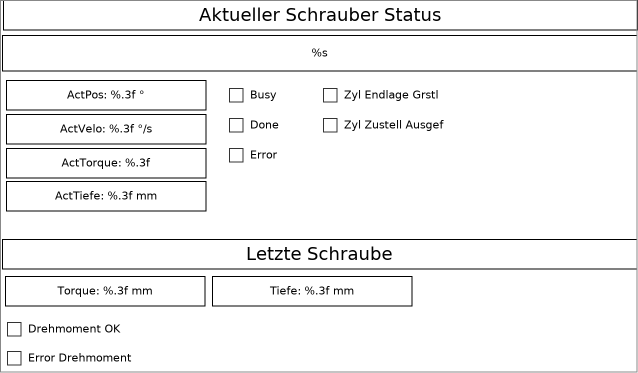
VISUALIZATION Frame_Schrauber_Status  // 638x373
VAR_IN_OUT
	sState	:STRING;
	
	bGrdstlgSchrEinh			: BOOL;
	bZustellZylAusgef			: BOOL;
	
	bBusy	:BOOL;
	bDone	:BOOL;
	bError	:BOOL;
	bErrorDrehmoment		:BOOL;
	bDrehmomentOk			:BOOL;
	nDrehmomentMw			:LREAL;	(* Drehmoment Mittelwert *)
	
	nActPos					:LREAL;
	nActVelo				:LREAL;
	nActTiefe				:LREAL;
	
	nDrehmomentLetzteSchr	:LREAL;	(* Drehmoment Letzte Schraubvorgang *)	
	nTiefeLetzteSchr		:LREAL;	(* Tiefe Letzte Schraubvorgang *)	
END_VAR
    Checkbox (227,80 150x30), "Busy", variable: bBusy, input disabled if: TRUE
    Checkbox (227,110 150x30), "Done", variable: bDone, input disabled if: TRUE
    Checkbox (227,140 150x30), "Error", variable: bError, input disabled if: TRUE
    RoundedRectangle (2,35 635x36), "%s", text variable: sState
    Checkbox (5,314 150x30), "Drehmoment OK", variable: bDrehmomentOk, input disabled if: TRUE
    Rectangle (6,80 200x30), "ActPos: %.3f °", text variable: nActPos
    Rectangle (6,114 200x30), "ActVelo: %.3f °/s", text variable: nActVelo
    Rectangle (6,148 200x30), "ActTorque: %.3f", text variable: nDrehmomentMw
    Rectangle (6,181 200x30), "ActTiefe: %.3f mm", text variable: nActTiefe
    Rectangle (212,276 200x30), "Tiefe: %.3f mm", text variable: nTiefeLetzteSchr
    Rectangle (5,276 200x30), "Torque: %.3f mm", text variable: nDrehmomentLetzteSchr
    Checkbox (5,343 150x30), "Error Drehmoment", variable: bErrorDrehmoment, input disabled if: TRUE
    Rectangle (3,0 635x30), "Aktueller Schrauber Status"
    Rectangle (2,239 635x30), "Letzte Schraube"
    Checkbox (321,80 150x30), "Zyl Endlage Grstl", variable: bGrdstlgSchrEinh, input disabled if: true
    Checkbox (321,110 150x30), "Zyl Zustell Ausgef", variable: bZustellZylAusgef, input disabled if: true
END_VISUALIZATION

(* stored: Version 1.1.0.1, ProductVersion 3.1.4024.15
   Visu Frame_Schrauber_Status: Id {0f763a79-15c5-42e5-8302-2fd114b4ed4a} *)
